(* IEC 61131-3 sources: test/src-senvion_wtt_fast-plc/InterTaskCommunication, 2 files *)

(* ---- GetHandles.st ---- *)
PROGRAM GetHandles
VAR CONSTANT
	NbrOfHandleBlocks 	: INT := 2;
END_VAR
VAR
	i 				: INT;
	ErrMsgDone		: BOOL;
END_VAR
VAR_OUTPUT
	InitDone		: BOOL;
END_VAR

i := i + 1;

IF(i > NbrOfHandleBlocks)THEN
	i :=1;
END_IF

(* -------------------------------------------------------------------------------------------- *)
(* --- Get handles from WTT_IO - program max. 10 handles in each block *)
(* -------------------------------------------------------------------------------------------- *)

CASE i OF
	1:
		Handles.Example1 := WTTL_GetPresHd(LogicalNodeName := 'WTUR', DataObjectName := 'Example1' , CalcPer := 0);

	2:
		Handles.Example2 := WTTL_GetPresHd(LogicalNodeName := 'WTUR', DataObjectName := 'Example2' , CalcPer := 0);

END_CASE

(* -------------------------------------------------------------------------------------------- *)
(* --- Check handles *)
(* -------------------------------------------------------------------------------------------- *)
IF	(Handles.Example1 <> 0) AND
	(Handles.Example2 <> 0)
THEN
	InitDone := TRUE;
END_IF

IF NOT(InitDone) AND NOT(ErrMsgDone) AND (i = NbrOfHandleBlocks) THEN
	Util_LogErr('Error during initialization of the handles for WTT_FAST');
	ErrMsgDone := TRUE;
END_IF

END_PROGRAM

(* ---- TaskComFast.st ---- *)
PROGRAM TaskComFast
VAR
	IntMainToFast			: MainToFast;
	IntFastToMain			: FastToMain;
	ChkCnt					: DINT;
	MainToFastChkCntErr		: DINT;

	Parameter1	   	: REAL;
	Parameter2		: REAL;
	Parameter3		: REAL;
	Parameter4		: REAL;

END_VAR

(* -------------------------------------------------------------------*)
(* -- Data from WTT_FAST to WTT_MAIN                                 --*)
(* -------------------------------------------------------------------*)
ChkCnt := ChkCnt + 1;

IntMainToFast.ChkCntStart 	:= ChkCnt;
IntFastToMain.Speed			:= 1500;
IntFastToMain.Status		:= TRUE;
IntMainToFast.ChkCntEnd 	:= ChkCnt;

Mem_AtomicCopy(Dst := ADR(FastToMain), Src := ADR(IntFastToMain), Len := SIZEOF(FastToMain));

(* -------------------------------------------------------------------*)
(* -- Data from WTT_MAIN  to WTT_FAST                                 --*)
(* -------------------------------------------------------------------*)

Mem_AtomicCopy(Dst := ADR(IntMainToFast), Src := ADR(MainToFast), Len := SIZEOF(MainToFast));

IF(IntMainToFast.ChkCntStart = IntMainToFast.ChkCntEnd)THEN
	Parameter1 := IntMainToFast.Parameter1;
	Parameter2 := IntMainToFast.Parameter2;
	Parameter3 := IntMainToFast.Parameter3;
	Parameter4 := IntMainToFast.Parameter4;
ELSE
	MainToFastChkCntErr := MainToFastChkCntErr + 1;
END_IF

END_PROGRAM
